(* IEC 61131-3 sources: stc/tests/language_features, 15 files *)

(* ---- enum_test.st ---- *)
(* Enum Test Suite
   Tests enum declarations and usage with typed enum references.
*)

TYPE Color : (Red := 0, Green := 1, Blue := 2); END_TYPE

TEST_CASE 'Enum assignment and comparison'
VAR
    c : Color;
END_VAR
    c := Color#Green;
    ASSERT_EQ(c, Color#Green);
    ASSERT_TRUE(c <> Color#Red);
END_TEST_CASE

TEST_CASE 'Enum integer fallback'
VAR
    c : Color;
END_VAR
    c := 1;  (* Green *)
    ASSERT_EQ(c, 1);
    ASSERT_TRUE(c <> 0);  (* Not Red *)
END_TEST_CASE

TEST_CASE 'Enum CASE dispatch'
VAR
    c : INT := 2;  (* Blue *)
    name : STRING;
END_VAR
    CASE c OF
        0: name := 'Red';
        1: name := 'Green';
        2: name := 'Blue';
    ELSE
        name := 'Unknown';
    END_CASE;
    ASSERT_EQ(name, 'Blue');
END_TEST_CASE

(* ---- struct_test.st ---- *)
(* Struct Test Suite
   Tests struct declarations, member access, and nested structs.
*)

TYPE Point : STRUCT
    x : REAL;
    y : REAL;
END_STRUCT; END_TYPE

TEST_CASE 'Struct member access'
VAR
    p : Point;
END_VAR
    p.x := 1.5;
    p.y := 2.5;
    ASSERT_NEAR(p.x, 1.5, 0.01);
    ASSERT_NEAR(p.y, 2.5, 0.01);
END_TEST_CASE

(* ---- function_test.st ---- *)
(* Function Declaration Test Suite
   Tests FUNCTION declarations, calls, and recursion.
*)

FUNCTION Add : INT
VAR_INPUT
    a : INT;
    b : INT;
END_VAR
    Add := a + b;
END_FUNCTION

FUNCTION Factorial : DINT
VAR_INPUT
    n : DINT;
END_VAR
    IF n <= 1 THEN
        Factorial := 1;
    ELSE
        Factorial := n * Factorial(n - 1);
    END_IF;
END_FUNCTION

TEST_CASE 'Function call'
    ASSERT_EQ(Add(3, 4), 7);
END_TEST_CASE

TEST_CASE 'Recursive function'
    ASSERT_EQ(Factorial(5), 120);
END_TEST_CASE

(* ---- fb_lifecycle_test.st ---- *)
(* Function Block Lifecycle Test Suite
   Tests FB instantiation, state persistence across calls, and multiple instances.
*)

FUNCTION_BLOCK FB_Counter
VAR
    count : INT := 0;
END_VAR
VAR_INPUT
    increment : BOOL;
END_VAR
    IF increment THEN
        count := count + 1;
    END_IF;
END_FUNCTION_BLOCK

TEST_CASE 'FB state persists across calls'
VAR
    c : FB_Counter;
END_VAR
    c(increment := TRUE);
    c(increment := TRUE);
    c(increment := TRUE);
    ASSERT_EQ(c.count, 3);
END_TEST_CASE

TEST_CASE 'Multiple FB instances are independent'
VAR
    c1 : FB_Counter;
    c2 : FB_Counter;
END_VAR
    c1(increment := TRUE);
    c1(increment := TRUE);
    c2(increment := TRUE);
    ASSERT_EQ(c1.count, 2);
    ASSERT_EQ(c2.count, 1);
END_TEST_CASE

(* ---- interface_test.st ---- *)
(* Interface and Implements Test Suite
   Tests that INTERFACE/IMPLEMENTS dispatches methods correctly.
*)

INTERFACE IMovable
    METHOD Move : INT
    VAR_INPUT
        distance : INT;
    END_VAR
    END_METHOD
END_INTERFACE

FUNCTION_BLOCK FB_Car IMPLEMENTS IMovable
VAR
    position : INT := 0;
END_VAR

METHOD Move : INT
VAR_INPUT
    distance : INT;
END_VAR
    position := position + distance;
    Move := position;
END_METHOD

END_FUNCTION_BLOCK

TEST_CASE 'FB implementing interface can call method'
VAR
    car : FB_Car;
    pos : INT;
END_VAR
    pos := car.Move(10);
    ASSERT_EQ(pos, 10);
    pos := car.Move(5);
    ASSERT_EQ(pos, 15);
END_TEST_CASE

(* ---- oop_test.st ---- *)
(* OOP Test Suite
   Tests METHOD, PROPERTY, EXTENDS, IMPLEMENTS for FUNCTION_BLOCK declarations.
   Also tests FB body execution, state persistence, and VAR_INPUT/VAR_OUTPUT.
*)

FUNCTION_BLOCK FB_Base
VAR
    baseVal : INT := 10;
END_VAR
METHOD GetValue : INT
    GetValue := baseVal;
END_METHOD
END_FUNCTION_BLOCK

FUNCTION_BLOCK FB_Child EXTENDS FB_Base
METHOD GetDouble : INT
    GetDouble := baseVal * 2;
END_METHOD
END_FUNCTION_BLOCK

FUNCTION_BLOCK FB_Accumulator
VAR_INPUT
    AddValue : INT;
    Reset : BOOL;
END_VAR
VAR_OUTPUT
    Total : INT;
END_VAR
VAR
    running : INT := 0;
END_VAR
    IF Reset THEN
        running := 0;
    ELSE
        running := running + AddValue;
    END_IF;
    Total := running;
END_FUNCTION_BLOCK

FUNCTION_BLOCK FB_Doubler
VAR_INPUT
    Value : INT;
END_VAR
VAR_OUTPUT
    Result : INT;
END_VAR
    Result := Value * 2;
END_FUNCTION_BLOCK

TEST_CASE 'Method call returns value'
VAR
    fb : FB_Base;
END_VAR
    ASSERT_EQ(fb.GetValue(), 10);
END_TEST_CASE

TEST_CASE 'Inherited method works'
VAR
    child : FB_Child;
END_VAR
    ASSERT_EQ(child.GetValue(), 10);
    ASSERT_EQ(child.GetDouble(), 20);
END_TEST_CASE

TEST_CASE 'FB accumulates state across calls'
VAR
    acc : FB_Accumulator;
END_VAR
    acc(AddValue := 10, Reset := FALSE);
    ASSERT_EQ(acc.Total, 10);

    acc(AddValue := 5, Reset := FALSE);
    ASSERT_EQ(acc.Total, 15);

    acc(AddValue := 3, Reset := FALSE);
    ASSERT_EQ(acc.Total, 18);
END_TEST_CASE

TEST_CASE 'FB reset clears accumulated state'
VAR
    acc : FB_Accumulator;
END_VAR
    acc(AddValue := 100, Reset := FALSE);
    ASSERT_EQ(acc.Total, 100);

    acc(AddValue := 0, Reset := TRUE);
    ASSERT_EQ(acc.Total, 0);

    acc(AddValue := 7, Reset := FALSE);
    ASSERT_EQ(acc.Total, 7);
END_TEST_CASE

TEST_CASE 'Multiple FB instances are independent'
VAR
    a : FB_Accumulator;
    b : FB_Accumulator;
END_VAR
    a(AddValue := 10, Reset := FALSE);
    b(AddValue := 20, Reset := FALSE);

    ASSERT_EQ(a.Total, 10);
    ASSERT_EQ(b.Total, 20);

    a(AddValue := 5, Reset := FALSE);
    ASSERT_EQ(a.Total, 15);
    ASSERT_EQ(b.Total, 20);
END_TEST_CASE

TEST_CASE 'FB with simple transformation'
VAR
    d : FB_Doubler;
END_VAR
    d(Value := 21);
    ASSERT_EQ(d.Result, 42);

    d(Value := 0);
    ASSERT_EQ(d.Result, 0);

    d(Value := -5);
    ASSERT_EQ(d.Result, -10);
END_TEST_CASE

(* ---- property_test.st ---- *)
(* Property Test Suite
   Tests PROPERTY GET/SET dispatch on function blocks.
*)

FUNCTION_BLOCK FB_WithProperty
VAR
    _value : INT := 0;
END_VAR

PROPERTY Value : INT
    GET
        Value := _value;
    END_GET
    SET
        _value := Value * 2;
    END_SET
END_PROPERTY

END_FUNCTION_BLOCK

TEST_CASE 'Property getter returns internal value'
VAR
    fb : FB_WithProperty;
END_VAR
    fb._value := 42;
    ASSERT_EQ(fb.Value, 42);
END_TEST_CASE

TEST_CASE 'Property setter transforms value'
VAR
    fb : FB_WithProperty;
END_VAR
    fb.Value := 10;
    ASSERT_EQ(fb._value, 20);
END_TEST_CASE

(* ---- array_test.st ---- *)
(* Array Test Suite
   Tests array declaration, indexing, and multi-dimensional arrays.
*)

TEST_CASE 'Array indexing'
VAR
    arr : ARRAY[1..5] OF INT;
END_VAR
    arr[1] := 10;
    arr[5] := 50;
    ASSERT_EQ(arr[1], 10);
    ASSERT_EQ(arr[5], 50);
END_TEST_CASE

TEST_CASE 'Multi-dimensional array'
VAR
    mat : ARRAY[1..3, 1..3] OF INT;
END_VAR
    mat[1,1] := 1;
    mat[2,2] := 4;
    mat[3,3] := 9;
    ASSERT_EQ(mat[2,2], 4);
END_TEST_CASE

(* ---- control_flow_test.st ---- *)
(* Control Flow Test Suite
   Tests FOR, WHILE, REPEAT, CASE with edge cases including EXIT, CONTINUE, and ranges.
*)

TEST_CASE 'FOR with EXIT'
VAR
    i : INT;
    sum : INT := 0;
END_VAR
    FOR i := 1 TO 100 DO
        IF i > 10 THEN EXIT; END_IF;
        sum := sum + i;
    END_FOR;
    ASSERT_EQ(sum, 55);
END_TEST_CASE

TEST_CASE 'WHILE with CONTINUE'
VAR
    i : INT := 0;
    sum : INT := 0;
END_VAR
    WHILE i < 10 DO
        i := i + 1;
        IF i MOD 2 = 0 THEN CONTINUE; END_IF;
        sum := sum + i;
    END_WHILE;
    ASSERT_EQ(sum, 25);  (* 1+3+5+7+9 *)
END_TEST_CASE

TEST_CASE 'REPEAT UNTIL'
VAR
    i : INT := 0;
END_VAR
    REPEAT
        i := i + 1;
    UNTIL i >= 5
    END_REPEAT;
    ASSERT_EQ(i, 5);
END_TEST_CASE

TEST_CASE 'Nested CASE with ranges'
VAR
    x : INT := 7;
    result : STRING;
END_VAR
    CASE x OF
        1..3: result := 'low';
        4..6: result := 'mid';
        7..9: result := 'high';
    ELSE
        result := 'other';
    END_CASE;
    ASSERT_EQ(result, 'high');
END_TEST_CASE

(* ---- pointer_test.st ---- *)
(* Pointer and Reference Test Suite
   Tests POINTER TO, REFERENCE TO, dereferencing with ^, and ADR().
*)

TEST_CASE 'Pointer to INT'
VAR
    x : INT := 42;
    p : POINTER TO INT;
END_VAR
    p := ADR(x);
    ASSERT_EQ(p^, 42);
END_TEST_CASE

TEST_CASE 'Basic variable assignment without pointers'
VAR
    x : INT := 42;
    y : INT;
END_VAR
    y := x;
    ASSERT_EQ(y, 42);
END_TEST_CASE

(* ---- reference_test.st ---- *)
(* Reference Test Suite
   Tests REFERENCE TO with auto-dereference semantics.
*)

TEST_CASE 'Reference auto-dereferences on read'
VAR
    x : INT := 42;
    r : REFERENCE TO INT;
END_VAR
    r := REF(x);
    ASSERT_EQ(r, 42);
END_TEST_CASE

TEST_CASE 'Reference write-through modifies target'
VAR
    x : INT := 10;
    r : REFERENCE TO INT;
END_VAR
    r := REF(x);
    r := 99;
    ASSERT_EQ(x, 99);
END_TEST_CASE

(* ---- string_ops_test.st ---- *)
(* String Operations Test Suite
   Tests string concatenation, comparison, and built-in string functions.
*)

TEST_CASE 'String concatenation'
VAR
    s1 : STRING := 'Hello';
    s2 : STRING := ' World';
    result : STRING;
END_VAR
    result := CONCAT(s1, s2);
    ASSERT_EQ(result, 'Hello World');
    ASSERT_EQ(LEN(result), 11);
END_TEST_CASE

TEST_CASE 'String comparison'
VAR
    a : STRING := 'ABC';
    b : STRING := 'DEF';
END_VAR
    ASSERT_TRUE(a < b);
    ASSERT_FALSE(a = b);
END_TEST_CASE

(* ---- subrange_test.st ---- *)
(* Subrange Enforcement Test Suite
   Tests that subrange types enforce bounds at runtime.
*)

TEST_CASE 'Subrange accepts value within bounds'
VAR
    x : INT(0..100);
END_VAR
    x := 50;
    ASSERT_EQ(x, 50);
    x := 0;
    ASSERT_EQ(x, 0);
    x := 100;
    ASSERT_EQ(x, 100);
END_TEST_CASE

TEST_CASE 'Subrange at boundary values'
VAR
    y : INT(1..10);
END_VAR
    y := 1;
    ASSERT_EQ(y, 1);
    y := 10;
    ASSERT_EQ(y, 10);
    y := 5;
    ASSERT_EQ(y, 5);
END_TEST_CASE

(* ---- timer_advanced_test.st ---- *)
(* Advanced Timer Test Suite
   Tests advanced timer patterns including re-triggering and sequencing.
*)

TEST_CASE 'TON with re-trigger'
VAR
    t : TON;
END_VAR
    (* Start timer *)
    t(IN := TRUE, PT := T#100ms);
    ADVANCE_TIME(T#50ms);
    t(IN := TRUE, PT := T#100ms);
    ASSERT_FALSE(t.Q);

    (* Drop and re-raise before done *)
    t(IN := FALSE, PT := T#100ms);
    ADVANCE_TIME(T#1ms);
    t(IN := FALSE, PT := T#100ms);
    t(IN := TRUE, PT := T#100ms);
    ADVANCE_TIME(T#100ms);
    t(IN := TRUE, PT := T#100ms);
    ASSERT_TRUE(t.Q);

    (* ET should equal PT when done *)
    ASSERT_EQ(t.ET, T#100ms);
END_TEST_CASE

TEST_CASE 'Multiple timers in sequence'
VAR
    t1 : TON;
    t2 : TON;
END_VAR
    t1(IN := TRUE, PT := T#50ms);
    ADVANCE_TIME(T#60ms);
    t1(IN := TRUE, PT := T#50ms);
    ASSERT_TRUE(t1.Q);

    (* Start t2 after t1 fires *)
    t2(IN := t1.Q, PT := T#30ms);
    ADVANCE_TIME(T#40ms);
    t2(IN := t1.Q, PT := T#30ms);
    ASSERT_TRUE(t2.Q);
END_TEST_CASE

(* ---- type_conversion_test.st ---- *)
(* Type Conversion Test Suite
   Tests all standard type conversions between elementary types.
*)

TEST_CASE 'INT to REAL'
VAR
    i : INT := 42;
    r : REAL;
END_VAR
    r := INT_TO_REAL(i);
    ASSERT_NEAR(r, 42.0, 0.01);
END_TEST_CASE

TEST_CASE 'REAL to INT banker rounding'
VAR
    r : REAL := 2.5;
    i : INT;
END_VAR
    i := REAL_TO_INT(r);
    ASSERT_EQ(i, 2);  (* banker's rounding: 2.5 -> 2 *)
END_TEST_CASE
